# B&R Automation Studio project CaseWeek_user
Automation Studio 4.9.3.144 SP; technology packages: mappView 5.14.2

## Configuration X20CP1584

CPU X20CP1584, AutomationRuntime C4.90, Build 4.1.2, Safety 0.0, Vc V4.34.3

### Task classes (Cpu.sw)
```
Cyclic#1:
  ClockSigna <- Wizualizacja.ClockSignal.prg
Cyclic#4:
  Tanks <- Sterowanie.Tanks.prg
Libraries: standard
```

### Hardware
```
X20CP1584 : X20CP1584 v1.8.1.0
  Connector IF2:
    ActivateDevice = 1
  Connector IF3:
    DNAConfiguration = manual
  ConfigurationID = CaseWeek_user_X20CP1584
  Simulation = 1
  ActivateOpcUa = 1
  OpcUaInformationModels_PV_Version = 1
```

## Logical view

Binary libraries used (declarations not repeated): operator, runtime, astime, AsIecCon, standard


### Program Logical/Wizualizacja/ClockSignal (IEC)

#### Variables.var
```iecst
VAR
	Clock : BOOL;
	ClockStatus : USINT;
	Mixer : BOOL;
	MixerStatus : USINT;
	TON_1 : TON;
	TON_0 : TON;
END_VAR
```

#### Main.st
```iecst
PROGRAM _INIT
END_PROGRAM

PROGRAM _CYCLIC
	CASE ClockStatus OF
		0:
			TON_1.IN:=TRUE;
			Clock:=TRUE;
			IF TON_1.Q THEN
				ClockStatus:=1;
				TON_1.IN:=FALSE;
			END_IF
		1:
			Clock:=FALSE;
			TON_1.IN:=TRUE;
			IF TON_1.Q THEN
				TON_1.IN:=FALSE;
				ClockStatus:=0;
			END_IF;
	END_CASE

	CASE MixerStatus OF
		0:
			TON_0.IN:=TRUE;
			Mixer:=TRUE;
			IF TON_0.Q THEN
				MixerStatus:=1;
				TON_0.IN:=FALSE;
			END_IF
		1:
			Mixer:=FALSE;
			TON_0.IN:=TRUE;
			IF TON_0.Q THEN
				TON_0.IN:=FALSE;
				MixerStatus:=0;
			END_IF;
	END_CASE

	TON_1(PT:=T#150ms);
	TON_0 (PT:=T#500ms);
END_PROGRAM

PROGRAM _EXIT
	(* Insert code here *)

END_PROGRAM
```

- Visualisation Logical/mappView (not shown)

### mappingVariables.var
```iecst
(*Zmienne które sa uzywane przez symulacje. Nalezy je przypisac do zmiennych w programie sterujacym*)
VAR
	gZb1_poziom : INT; (*Poziom cieczy w zbiorniku 1*)
	gZb2_poziom : INT; (*Poziom cieczy w zbiorniku 2*)
	gZb3_poziom : INT; (*Poziom cieczy w zbiorniku 3*)
	gZb1_zawor : BOOL; (*0 - zawor zamkniety, 1 - zawor otwarty*)
	gZb2_zawor : BOOL; (*0 - zawor zamkniety, 1 - zawor otwarty*)
	gZb3_zawor_lewy : INT; (*% otwarcia zaworu lewego (0-100)*)
	gZb3_zawor_prawy : INT; (*% otwarcia zaworu prawego (0-100)*)
	gZb3_zawor_glowny : BOOL; (*0 - zawor zamkniety, 1 - zawor otwarty*)
	gMieszadlo : BOOL; (*0 - mieszadlo wylaczone, 1- mieszadlo wlaczone*)
END_VAR
```

### Program Logical/Sterowanie/Tanks (IEC)

#### Main.st - Init, cyclic, exit code
```iecst
PROGRAM _INIT
	gZb1_poziom;
	gZb1_zawor;
	gZb2_poziom;
	gZb2_zawor;

	gZb3_poziom;
	gZb3_zawor_glowny;
	gZb3_zawor_lewy;
	gZb3_zawor_prawy;

	ManualControl;

	gMieszadlo;

	gTanks.Loop := TRUE;

	gTanks.StirTime := T#5s;
	gTanks.EnableStir := TRUE;

	gTanks.FirstTankCapacity := 10000;
	gTanks.SecondTankCapacity := 10000;
	gTanks.MainTankCapacity := 10000;

	gTanks.FirstTankMaxLevel := 8000;
	gTanks.SecondTankMaxLevel := 8000;
	gTanks.MainTankMaxLevel := 8000;
	gTanks.MainTankMinLevel := 0;

	FirstValveOpenLevel := 100;
	SecondValveOpenLevel := 100;

	gTanks.CurrentState := TANKS_STOP;

	TON_Stir();

	FirstRun := FALSE;

END_PROGRAM

PROGRAM _CYCLIC

	IF gTanks.Stop THEN
		gTanks.CurrentState := TANKS_STOP;
	END_IF

	IF gTanks.EnableStir THEN
		gTanks.MainTankMaxLevel := 10000;
	ELSE
		gTanks.MainTankMaxLevel := 8000;
	END_IF

	CASE gTanks.CurrentState OF
		TANKS_STOP:
			gTanks.FirstTankFilled := FALSE;
			gTanks.SecondTankFilled := FALSE;
			gTanks.MainTankFilled := FALSE;
			TON_Stir.IN := FALSE;

			Status := 0;

			IF gTanks.Start THEN
				gTanks.CurrentState := TANKS_FILL_SUB;
			END_IF

		TANKS_FILL_SUB:
			Status := 1;
			IF gZb1_poziom>=gTanks.FirstTankMaxLevel THEN
				gZb1_zawor := FALSE;
				gTanks.FirstTankFilled := TRUE;
			ELSIF NOT gTanks.FirstTankFilled THEN
				gZb1_zawor := TRUE;
			END_IF

			IF gZb2_poziom>=gTanks.SecondTankMaxLevel THEN
				gZb2_zawor := FALSE;
				gTanks.SecondTankFilled := TRUE;
			ELSIF NOT gTanks.SecondTankFilled THEN
				gZb2_zawor := TRUE;
			END_IF

			IF gTanks.FirstTankFilled AND gTanks.SecondTankFilled THEN
				gTanks.CurrentState := TANKS_FILL_MAIN;
			END_IF

		TANKS_FILL_MAIN:
			IF gZb3_poziom >= gTanks.MainTankMaxLevel THEN
				gZb3_zawor_lewy := 0;
				gZb3_zawor_prawy := 0;
				gTanks.MainTankFilled := TRUE;
			ELSE
				gZb3_zawor_glowny := FALSE;
				gZb3_zawor_lewy := SecondValveOpenLevel;
				gZb3_zawor_prawy := FirstValveOpenLevel;
			END_IF

			IF gTanks.MainTankFilled THEN
				IF gTanks.EnableStir THEN
					gTanks.CurrentState := TANKS_STIR;
				ELSE
					gTanks.CurrentState := TANKS_DRAIN_MAIN;
				END_IF
			END_IF

		TANKS_STIR:
			TON_Stir.IN := TRUE;
			IF TON_Stir.Q THEN
				gTanks.CurrentState := TANKS_DRAIN_MAIN;
				gMieszadlo := 0;
				TON_Stir.IN := FALSE;
			ELSE
				gMieszadlo := 1;
			END_IF

		TANKS_DRAIN_MAIN:
			IF gZb3_poziom <= gTanks.MainTankMinLevel THEN
				gZb3_zawor_glowny := FALSE;
				gTanks.CurrentState := TANKS_STOP;
			ELSE
				gZb3_zawor_glowny := TRUE;
			END_IF

	END_CASE

	TON_Stir(PT := gTanks.StirTime);

END_PROGRAM

PROGRAM _EXIT
	gTanks.MainTankFilled := FALSE;
	gTanks.FirstTankFilled := FALSE;
	gTanks.SecondTankFilled := FALSE;
	gZb1_zawor := FALSE;
	gZb2_zawor := FALSE;
	gZb3_zawor_glowny := FALSE;
	gZb3_zawor_lewy := 0;
	gZb3_zawor_prawy := 0;
	gMieszadlo := FALSE;

END_PROGRAM
```

#### Types.typ - Local data types
```iecst
TYPE
	TanksPara : 	STRUCT  (*Parameters used to define gTanks*)
		Stop : BOOL; (*Stops the state machine*)
		Start : BOOL; (*Starts the state machine*)
		Loop : BOOL; (*Enables closed loop execution*)
		EnableStir : BOOL; (*Enables stirring*)
		StirTime : TIME; (*Defines stirring time*)
		FirstTankFilled : BOOL; (*Has the first subsidiary tank been filled to set level?*)
		SecondTankFilled : BOOL; (*Has the second subsidiary tank been filled to set level?*)
		MainTankFilled : BOOL; (*Has the main tank been filled to set level?*)
		FirstTankMaxLevel : INT; (*Defines desired fill level for the first tank*)
		SecondTankMaxLevel : INT; (*Defines desired fill level for the second tank*)
		MainTankMaxLevel : INT; (*Defines desired fill level for the main tank*)
		MainTankMinLevel : INT; (*Defines the minimum allowed fill level for the main tank*)
		FirstTankCapacity : INT; (*Defines first tank's capacity*)
		SecondTankCapacity : INT; (*Defines second tank's capacity*)
		MainTankCapacity : INT; (*Defines main tank's capacity*)
		CurrentState : TanksStateMachine; (*Defines which state the machine is in*)
	END_STRUCT;
	TanksStateMachine :
		( (*Main state machine used to define gTanks behaviour*)
		TANKS_FILL_SUB, (*Filling subsidiary tanks*)
		TANKS_FILL_MAIN, (*Filling main tank*)
		TANKS_STIR, (*Stirring main tank's contents*)
		TANKS_DRAIN_MAIN, (*Draining main tank*)
		TANKS_STOP (*All operation is stopped*)
		);
END_TYPE
```

#### Variables.var - Local variables
```iecst
VAR
	TON_Stir : TON;
	gTanks : TanksPara;
	FirstValveOpenLevel : INT;
	SecondValveOpenLevel : INT;
	FirstRun : BOOL;
	Status : USINT;
	ManualControl : BOOL;
END_VAR
```

Listed in the project but not available here: Logical/Global.typ, Logical/Global.var
